(*
Status information for a cabinet, will not change from cabinet to cabinet,
input/output represents bits 00-15 in safety controller.
*)
TYPE ST_MCCStatus :
STRUCT
    In: ST_MCCStatusIn;
    Out: ST_MCCStatusOut;
END_STRUCT
END_TYPE

(* stored: Version 1.1.0.1
   DUT ST_MCCStatus: Id {00ac038e-aa81-4175-9c09-5cd4fbc6f3e8} *)
